// TIA Portal project "Betriebsstundenzähler_KOP" (V16)

(* hardware
DEVICE "S7-1200 station_1"  S7-1200 Station
   slot 0: "Rack_0"  S7-1200 Rack  Rack  V1.0
   slot 1: "PLC_1"  CPU 1212C DC/DC/DC  6ES7 212-1AE40-0XB0  V4.4
*)

// ===== PLC "PLC_1"  CPU 1212C DC/DC/DC =====

VAR_GLOBAL   // PLC tag table "Default tag table"
   "Einschalttaste_Eingang" AT %I0.0 : Bool;
   "Resettaste_Eingang" AT %I0.1 : Bool;
   "Systemeinschalt_Bit" AT %M0.0 : Bool;
   "Reset_Bit" AT %M0.1 : Bool;
   "Sekunden_S" AT %MW4 : Int;
   "Sekunden_mS" AT %MD6 : DInt;
   "Minuten" AT %MW2 : Int;
   "Stunden" AT %MW10 : Int;
   "Stunden*1000" AT %MW12 : Int;
END_VAR

DATA_BLOCK "IO_DB"   // DB1
{ S7_Optimized_Access := 'TRUE' }
VERSION : 0.1
// stored: InstanceOfName IO
"IO"
BEGIN
END_DATA_BLOCK

DATA_BLOCK "Steuerlogik_DB"   // DB5
{ S7_Optimized_Access := 'TRUE' }
VERSION : 0.1
// stored: InstanceOfName Steuerlogik
"Steuerlogik"
BEGIN
END_DATA_BLOCK

// folder: System blocks/Program resources

DATA_BLOCK "Stunden_Zähler"   // DB2
{ S7_Optimized_Access := 'TRUE' }
AUTHOR : Simatic
FAMILY : IEC
NAME : CNTR
VERSION : 1.0
// stored: InstanceOfName IEC_COUNTER
"IEC_COUNTER"
BEGIN
END_DATA_BLOCK

DATA_BLOCK "Timer"   // DB3
{ S7_Optimized_Access := 'TRUE' }
AUTHOR : Simatic
FAMILY : IEC
NAME : IEC_TMR
VERSION : 1.0
// stored: InstanceOfName IEC_TIMER
"IEC_TIMER"
BEGIN
END_DATA_BLOCK

DATA_BLOCK "Minuten_Zähler"   // DB4
{ S7_Optimized_Access := 'TRUE' }
AUTHOR : Simatic
FAMILY : IEC
NAME : CNTR
VERSION : 1.0
// stored: InstanceOfName IEC_COUNTER
"IEC_COUNTER"
BEGIN
END_DATA_BLOCK

DATA_BLOCK "Stunden*1000_Zähler"   // DB6
{ S7_Optimized_Access := 'TRUE' }
AUTHOR : Simatic
FAMILY : IEC
NAME : CNTR
VERSION : 1.0
// stored: InstanceOfName IEC_COUNTER
"IEC_COUNTER"
BEGIN
END_DATA_BLOCK

// folder: (top level)

FUNCTION_BLOCK "IO"   // FB1, LAD
{ S7_Optimized_Access := 'TRUE' }
VERSION : 0.1
BEGIN

REGION Network 1
   // Eingänge
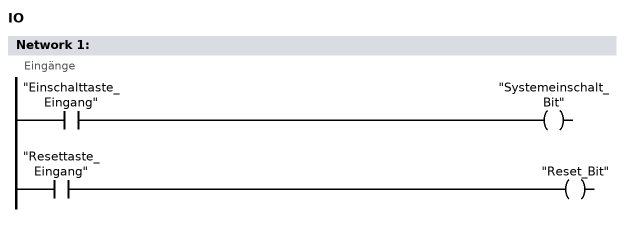
   RUNG wire#powerrail
      Contact( "Einschalttaste_Eingang" )
      Coil( "Systemeinschalt_Bit" )
   END_RUNG
   RUNG wire#powerrail
      Contact( "Resettaste_Eingang" )
      Coil( "Reset_Bit" )
   END_RUNG
   // the same network as SCL:
   "Systemeinschalt_Bit" := "Einschalttaste_Eingang";
   "Reset_Bit" := "Resettaste_Eingang";
END_REGION
END_FUNCTION_BLOCK

FUNCTION_BLOCK "Steuerlogik"   // FB2, LAD
{ S7_Optimized_Access := 'TRUE' }
VERSION : 0.1
   VAR
      Sekunden_mS : Int;
      Sekunden_mS_1 : Int;
      Minuten_ZählerDone_Bit : Bool;
      Stunden_ZählerDone_Bit : Bool;
      TimerDone_Bit : Bool;
      "Stunden*1000_DoneBit" : Bool;
      ONS : Bool;
      Reset_All : Bool;
      Timer_Reset : Bool;
      Minuten_Reset : Bool;
      Stunden_Reset : Bool;
      "Stunden*1000_Reset" : Bool;
   END_VAR
   VAR_TEMP   // added for the SCL form of the ladder/FBD networks
      _w1 : Bool;
      _w2 : Bool;
   END_VAR
BEGIN

REGION Network 1
   // Steuerlogik für Sekunden
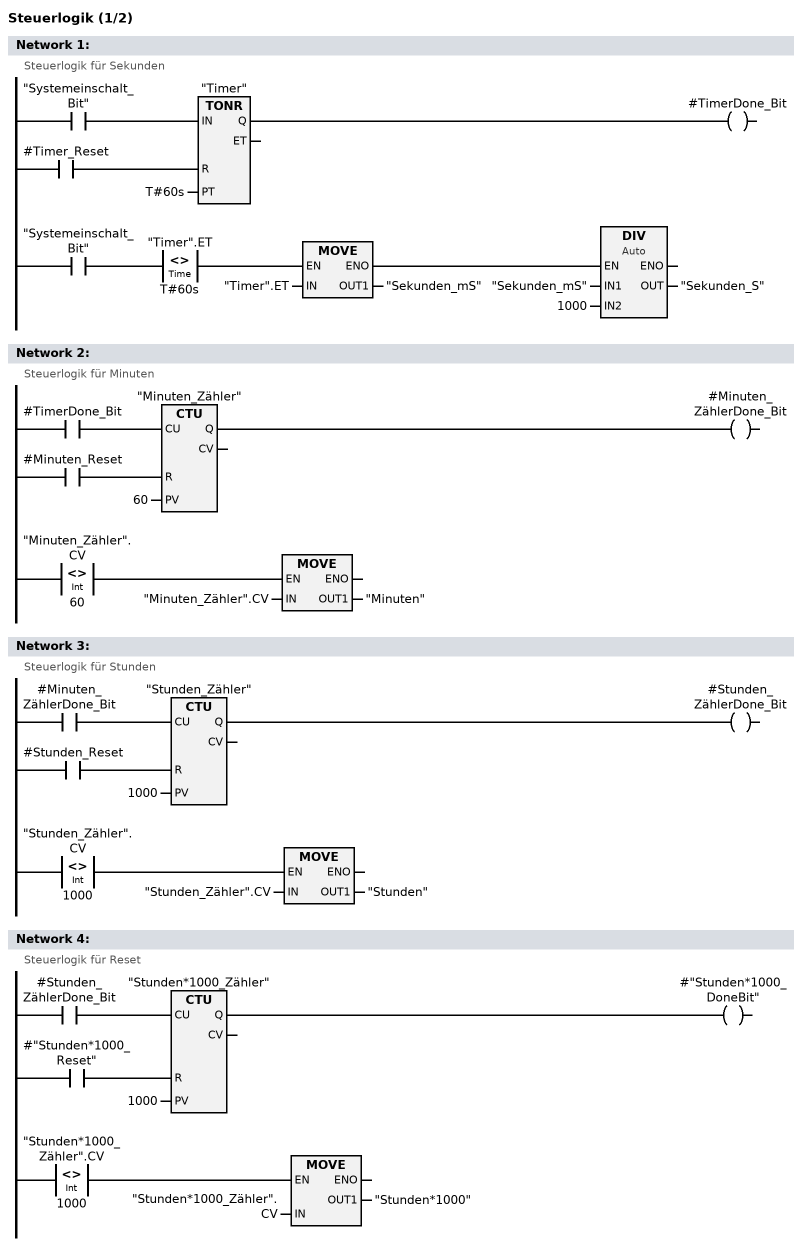
   "Timer".TONR(IN := "Systemeinschalt_Bit", R := #Timer_Reset, PT := T#60s);
   #TimerDone_Bit := "Timer".Q;
   IF "Systemeinschalt_Bit" AND ("Timer".ET <> T#60s) THEN
       "Sekunden_mS" := "Timer".ET;
       "Sekunden_S" := "Sekunden_mS" / 1000;
   END_IF;
END_REGION

REGION Network 2
   // Steuerlogik für Minuten
   "Minuten_Zähler".CTU(CU := #TimerDone_Bit, R := #Minuten_Reset, PV := 60);
   #Minuten_ZählerDone_Bit := "Minuten_Zähler".Q;
   IF "Minuten_Zähler".CV <> 60 THEN "Minuten" := "Minuten_Zähler".CV; END_IF;
END_REGION

REGION Network 3
   // Steuerlogik für Stunden
   "Stunden_Zähler".CTU(CU := #Minuten_ZählerDone_Bit, R := #Stunden_Reset, PV := 1000);
   #Stunden_ZählerDone_Bit := "Stunden_Zähler".Q;
   IF "Stunden_Zähler".CV <> 1000 THEN "Stunden" := "Stunden_Zähler".CV; END_IF;
END_REGION

REGION Network 4
   // Steuerlogik für Reset
   "Stunden*1000_Zähler".CTU(CU := #Stunden_ZählerDone_Bit, R := #"Stunden*1000_Reset", PV := 1000);
   #"Stunden*1000_DoneBit" := "Stunden*1000_Zähler".Q;
   IF "Stunden*1000_Zähler".CV <> 1000 THEN "Stunden*1000" := "Stunden*1000_Zähler".CV; END_IF;
END_REGION

REGION Network 5
   // Steuerlogik für Reset
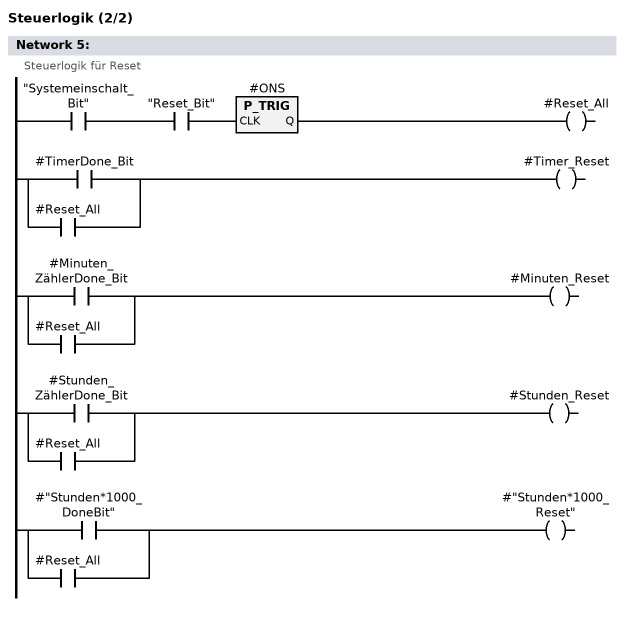
   RUNG wire#powerrail
      Contact( "Systemeinschalt_Bit" )
      Contact( "Reset_Bit" )
      P_Trig( #ONS )
      Coil( #Reset_All )
   END_RUNG
   RUNG wire#powerrail
      Contact( #TimerDone_Bit )
      wire#w1
      Coil( #Timer_Reset )
   END_RUNG
   RUNG wire#powerrail
      Contact( #Reset_All )
   END_RUNG wire#w1
   RUNG wire#powerrail
      Contact( #Minuten_ZählerDone_Bit )
      wire#w2
      Coil( #Minuten_Reset )
   END_RUNG
   RUNG wire#powerrail
      Contact( #Reset_All )
   END_RUNG wire#w2
   RUNG wire#powerrail
      Contact( #Stunden_ZählerDone_Bit )
      wire#w3
      Coil( #Stunden_Reset )
   END_RUNG
   RUNG wire#powerrail
      Contact( #Reset_All )
   END_RUNG wire#w3
   RUNG wire#powerrail
      Contact( #"Stunden*1000_DoneBit" )
      wire#w4
      Coil( #"Stunden*1000_Reset" )
   END_RUNG
   RUNG wire#powerrail
      Contact( #Reset_All )
   END_RUNG wire#w4
   // the same network as SCL:
   #_w1 := "Systemeinschalt_Bit" AND "Reset_Bit";
   #_w2 := #_w1 AND NOT #ONS;   // rising edge
   #ONS := #_w1;
   #Reset_All := #_w2;
   #Timer_Reset := #TimerDone_Bit OR #Reset_All;
   #Minuten_Reset := #Minuten_ZählerDone_Bit OR #Reset_All;
   #Stunden_Reset := #Stunden_ZählerDone_Bit OR #Reset_All;
   #"Stunden*1000_Reset" := #"Stunden*1000_DoneBit" OR #Reset_All;
END_REGION
END_FUNCTION_BLOCK

ORGANIZATION_BLOCK "Main"   // OB1, LAD, ProgramCycle
TITLE = "Main Program Sweep (Cycle)"
{ S7_Optimized_Access := 'TRUE' }
VERSION : 0.1
// PROJEKTBESCHREIBUNG:In diesem Projekt wird ein Steuerungssystem entwickelt, das die Laufzeit einer Hauptanlage erfasst. Sobald die Anlage eingeschaltet wird, beginnt der Zähler, die Betriebsdauer in Sekunden, Minuten, Hunderten und Tausenden von Stunden zu messen und in den Speicherregistern Sekunden_S, Minuten und Stunden abzulegen. Zusätzlich gibt es eine Reset-Taste, mit der der gesamte Zählerstand auf null zurückgesetzt werden kann, um eine neue Messung zu starten. Die Steuerung erfolgt über ein Einschalttaste. Solche Systeme sind essenziell, da Betriebsstunden oft als Grundlage für Wartung, Inspektion oder Garantieansprüche dienen.
// 
// TESTKRITERIEN:
// 1)Zum Starten: Führen Sie Ihr Programm in PLCSIM aus. "Sekunden_S","Minuten" und "Stunden" sollten alle auf Null stehen. Diese Werte sollten sich nicht bewegen.
// 
// 2)
// Als Nächstes erzwingen Sie den Einschalttaste_Eingang auf 1 (geschlossen). Nun sollten wir sehen, dass "Sekunden_S" akkumuliert. Es sollte immer wieder von 0 bis 59 zählen. Jedes Mal, wenn "Sekunden_S" eine Minute vollzählt, sollte "Minuten" um eins hochgehen. Irgendwann erreicht "Minuten" den Wert 59 und springt dann wieder selbst auf 0 zurück. Wenn das passiert, sollte "Stunden" um eins hochgehen. (Auch wenn wir es nicht so lange laufen lassen werden.) Nachdem "Stunden" den Wert 999 erreicht, sollte es wieder auf 0 zurückspringen und "Stunden*1000" um eins hochgehen. Und so weiter. Um zu testen, ob "Stunden" und "Stunden*1000" funktionieren, können Sie "Minuten" und "Stunden" manuell jeweils auf ihren Grenzwert setzen, um sicherzustellen, dass alles korrekt hochzählt.
// 3)
// 
// Drittens erzwingen Sie den Einschalttaste_Eingang wieder 0 (offen). Alle Ihre Akkumulatoren  sollten genau an der Stelle einfrieren, an der sie stehen.
// 
// 
// 4)Viertens erzwingen Sie den System-Run-Eingang ein letztes Mal auf 1 (geschlossen). Die Akkumulatoren sollten genau dort weiterzählen, wo sie aufgehört haben.
// 
// 
// 5)Schließlich schalten Sie Reset_Eingang EIN und dann wieder AUS. Alle Werten sollten alle auf 0 zurückgesetzt werden.
   VAR_INPUT
      Initial_Call : Bool;   // Initial call of this OB
      Remanence : Bool;   // =True, if remanent data are available
   END_VAR
BEGIN

REGION Network 1
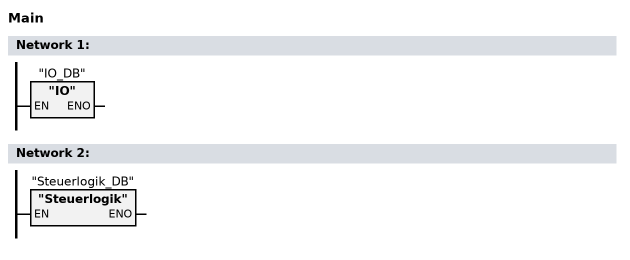
   RUNG wire#powerrail
      "IO_DB"()
   END_RUNG
   // the same network as SCL:
   "IO_DB"();   // "IO"
END_REGION

REGION Network 2
   RUNG wire#powerrail
      "Steuerlogik_DB"()
   END_RUNG
   // the same network as SCL:
   "Steuerlogik_DB"();   // "Steuerlogik"
END_REGION
END_ORGANIZATION_BLOCK